// TIA Portal V20 export
DATA_BLOCK "PM04"   // DB220
// stored: MemoryReserve 100
   VAR
      "C18 UNWINDER STOPPER FORWARD" : Bool;
      "C18 UNWINDER STOPPER BACKWARD" : Bool;
      "C19 UNWINDER DANCER FORWARD" : Bool;
      "C19 UNWINDER DANCER BACKWARD" : Bool;
      "C20 FEEDER CYLINDER DOWN" : Bool;
      "C20 FEEDER CYLINDER UP" : Bool;
      "C21 NG & MANUAL INPUT CYLINDER DOWN" : Bool;
      "C21 NG & MANUAL INPUT CYLINDER UP" : Bool;
      "C22 MAGAZINE LOCK CYLINDER UP" : Bool;
      "C22 MAGAZINE LOCK CYLINDER DOWN" : Bool;
      "C23 VISION PUSHER SUPPORT DOWN" : Bool;
      "C23 VISION PUSHER SUPPORT UP" : Bool;
      "C24 ELECTRODE NG BOX LOCK CYLINDER UP" : Bool;
      "C24 ELECTRODE NG BOX LOCK CYLINDER DOWN" : Bool;
      "C25 FRAME COVER FORWARD" : Bool;
      "C25 FRAME COVER BACKWARD" : Bool;
   END_VAR
BEGIN
END_DATA_BLOCK
